(* PLC project Tc2_Utilities.FB_AmsLogger Demo, tc3-libraries-kb TwinCAT 3.1 *)
(* stored: creationDateTime 2026-05-11T00:00:00, modificationDateTime 2026-05-11T00:00:00 *)

PROGRAM P_Demo_FB_AmsLogger
  VAR
    fbFB_AmsLogger : FB_AmsLogger;  (* FB_AmsLogger 实例 *)
    sNetId : T_AmsNetId := '';
    eMode : E_AmsLoggerMode := AMSLOGGER_RUN;
    sCfgFilePath : T_MaxString := '';
    bExecute : BOOL;
    tTimeout : TIME := DEFAULT_ADS_TIMEOUT;
    bBusy : BOOL;
    bError : BOOL;
    nErrId : UDINT;
  END_VAR

// =============================================================================
// 场景：老项目日志。
// 价值：兼容。
// 验证：调用 Add 加日志条目，目标日志服务应收到。
// 验证步骤：
//   1. 右键 PLC 项目 → Import PLCopenXML → 选本文件
//   2. 引用 Tc2_Utilities（References → Add library）
//   3. 编译 → 登录 → 运行；按上方『验证』行的指示在线写值观察
// =============================================================================

// 单次完整调用形式（所有 VAR_INPUT 显式赋值）
fbFB_AmsLogger(
    sNetId := sNetId,
    eMode := eMode,
    sCfgFilePath := sCfgFilePath,
    bExecute := bExecute,
    tTimeout := tTimeout,
    bBusy => bBusy,
    bError => bError,
    nErrId => nErrId
);
END_PROGRAM
